LIN {X 0,Y 241.644,Z 1084.792,A -85,B 0,C 180,E1 20729.307,E2 20729.307} C_VEL
LIN {X 0,Y 219.298,Z 1111.875,A -85,B 0,C 180,E1 20736.62,E2 20736.62} C_VEL
LIN {X 0,Y 200.143,Z 1133.56,A -85,B 0,C 180,E1 20746.024,E2 20746.024} C_VEL
LIN {X 0,Y 185.27,Z 1150.433,A -85,B 0,C 180,E1 20757.915,E2 20757.915} C_VEL
LIN {X 0,Y 177.934,Z 1160.639,A -85,B 0,C 180,E1 20770.102,E2 20770.102} C_VEL
LIN {X 0,Y 175.677,Z 1165.283,A -85,B 0,C 180,E1 20780.076,E2 20780.076} C_VEL
LIN {X 0,Y 175.749,Z 1166.865,A -85,B 0,C 180,E1 20790.002,E2 20790.002} C_VEL
LIN {X 0,Y 175.679,Z 1165.296,A -85,B 0,C 180,E1 20799.928,E2 20799.928} C_VEL
LIN {X 0,Y 179.088,Z 1158.782,A -85,B 0,C 180,E1 20812.714,E2 20812.714} C_VEL
LIN {X 0,Y 187.491,Z 1147.762,A -85,B 0,C 180,E1 20824.426,E2 20824.426} C_VEL
LIN {X 0,Y 202.393,Z 1131.049,A -85,B 0,C 180,E1 20835.333,E2 20835.333} C_VEL
LIN {X 0,Y 222.783,Z 1108.004,A -85,B 0,C 180,E1 20844.647,E2 20844.647} C_VEL
LIN {X 0,Y 229.425,Z 1100.179,A -85,B 0,C 180,E1 20846.96,E2 20846.96} C_VEL
LIN {X 0,Y 230.286,Z 1098.317,A -85,B 0,C 180,E1 20847.685,E2 20847.685} C_VEL
LIN {X 0,Y 210.353,Z 1100.814,A -85,B 0,C 180,E1 20854.414,E2 20854.414} C_VEL
LIN {X 0,Y 197.119,Z 1101.191,A -85,B 0,C 180,E1 20862.106,E2 20862.106} C_VEL
LIN {X 0,Y 189.812,Z 1096.992,A -85,B 0,C 180,E1 20884.573,E2 20884.573} C_VEL
LIN {X 0,Y 207.688,Z 1091.37,A -85,B 0,C 180,E1 20901.373,E2 20901.373} C_VEL
LIN {X 0,Y 233.869,Z 1084.178,A -85,B 0,C 180,E1 20911.188,E2 20911.188} C_VEL
LIN {X 0,Y 240.479,Z 1082.186,A -85,B 0,C 180,E1 20912.869,E2 20912.869} C_VEL
LIN {X 0,Y 238.937,Z 1085.101,A -85,B 0,C 180,E1 20913.875,E2 20913.875} C_VEL
LIN {X 0,Y 235.19,Z 1089.54,A -85,B 0,C 180,E1 20914.966,E2 20914.966} C_VEL
LIN {X 0,Y 223.73,Z 1099.969,A -85,B 0,C 180,E1 20917.059,E2 20917.059} C_VEL
LIN {X 0,Y 212.332,Z 1109.522,A -85,B 0,C 180,E1 20919.465,E2 20919.465} C_VEL
LIN {X 0,Y 191.319,Z 1129.897,A -85,B 0,C 180,E1 20929.672,E2 20929.672} C_VEL
LIN {X 0,Y 176.864,Z 1143.663,A -85,B 0,C 180,E1 20941.908,E2 20941.908} C_VEL
LIN {X 0,Y 169.807,Z 1151.224,A -85,B 0,C 180,E1 20954.482,E2 20954.482} C_VEL
LIN {X 0,Y 167.781,Z 1154.034,A -85,B 0,C 180,E1 20964.82,E2 20964.82} C_VEL
LIN {X 0,Y 167.899,Z 1154.368,A -85,B 0,C 180,E1 20969.998,E2 20969.998} C_VEL
LIN {X 0,Y 168.419,Z 1152.942,A -85,B 0,C 180,E1 20980.356,E2 20980.356} C_VEL
LIN {X 0,Y 173.955,Z 1146.544,A -85,B 0,C 180,E1 20994.1,E2 20994.1} C_VEL
LIN {X 0,Y 185.565,Z 1135.234,A -85,B 0,C 180,E1 21006.266,E2 21006.266} C_VEL
LIN {X 0,Y 204.238,Z 1117.516,A -85,B 0,C 180,E1 21017.059,E2 21017.059} C_VEL
LIN {X 0,Y 226.928,Z 1093.954,A -85,B 0,C 180,E1 21025.462,E2 21025.462} C_VEL
LIN {X 0,Y 249.884,Z 1066.331,A -85,B 0,C 180,E1 21031.468,E2 21031.468} C_VEL
LIN {X 0,Y 271.022,Z 1035.748,A -85,B 0,C 180,E1 21035.688,E2 21035.688} C_VEL
LIN {X 0,Y 281.025,Z 1018.475,A -85,B 0,C 180,E1 21037.454,E2 21037.454} C_VEL
LIN {X 0,Y 280.826,Z 1004.794,A -85,B 0,C 180,E1 21043.501,E2 21043.501} C_VEL
LIN {X 0,Y 280.116,Z 996.302,A -85,B 0,C 180,E1 21049.097,E2 21049.097} C_VEL
LIN {X 0,Y 279.786,Z 992.242,A -85,B 0,C 180,E1 21053.789,E2 21053.789} C_VEL
LIN {X 0,Y 279.873,Z 990.81,A -85,B 0,C 180,E1 21056.901,E2 21056.901} C_VEL
LIN {X 0,Y 279.882,Z 991.061,A -85,B 0,C 180,E1 21060.001,E2 21060.001} C_VEL
LIN {X 0,Y 279.944,Z 995.928,A -85,B 0,C 180,E1 21066.211,E2 21066.211} C_VEL
LIN {X 0,Y 280.603,Z 1005.561,A -85,B 0,C 180,E1 21072.465,E2 21072.465} C_VEL
LIN {X 0,Y 280.581,Z 1019.974,A -85,B 0,C 180,E1 21078.553,E2 21078.553} C_VEL
LIN {X 0,Y 260.028,Z 1054.145,A -85,B 0,C 180,E1 21082.426,E2 21082.426} C_VEL
LIN {X 0,Y 237.05,Z 1085.261,A -85,B 0,C 180,E1 21087.757,E2 21087.757} C_VEL
LIN {X 0,Y 213.909,Z 1112.152,A -85,B 0,C 180,E1 21095.059,E2 21095.059} C_VEL
LIN {X 0,Y 193.525,Z 1133.989,A -85,B 0,C 180,E1 21104.757,E2 21104.757} C_VEL
LIN {X 0,Y 178.365,Z 1150.132,A -85,B 0,C 180,E1 21116.513,E2 21116.513} C_VEL
LIN {X 0,Y 170.325,Z 1160.341,A -85,B 0,C 180,E1 21129.173,E2 21129.173} C_VEL
LIN {X 0,Y 167.809,Z 1164.992,A -85,B 0,C 180,E1 21139.606,E2 21139.606} C_VEL
LIN {X 0,Y 167.84,Z 1166.578,A -85,B 0,C 180,E1 21150.002,E2 21150.002} C_VEL
LIN {X 0,Y 167.811,Z 1165.005,A -85,B 0,C 180,E1 21160.399,E2 21160.399} C_VEL
LIN {X 0,Y 171.429,Z 1158.708,A -85,B 0,C 180,E1 21173.422,E2 21173.422} C_VEL
LIN {X 0,Y 180.75,Z 1147.459,A -85,B 0,C 180,E1 21185.904,E2 21185.904} C_VEL
LIN {X 0,Y 197.204,Z 1130.076,A -85,B 0,C 180,E1 21197.406,E2 21197.406} C_VEL
LIN {X 0,Y 218.094,Z 1107.676,A -85,B 0,C 180,E1 21206.423,E2 21206.423} C_VEL
LIN {X 0,Y 220.393,Z 1105.118,A -85,B 0,C 180,E1 21207.202,E2 21207.202} C_VEL
LIN {X 0,Y 220.637,Z 1103.734,A -85,B 0,C 180,E1 21207.988,E2 21207.988} C_VEL
LIN {X 0,Y 197.119,Z 1105.708,A -85,B 0,C 180,E1 21217.415,E2 21217.415} C_VEL
LIN {X 0,Y 183.691,Z 1104.522,A -85,B 0,C 180,E1 21230.51,E2 21230.51} C_VEL
LIN {X 0,Y 195.152,Z 1097.977,A -85,B 0,C 180,E1 21258.076,E2 21258.076} C_VEL
LIN {X 0,Y 224.215,Z 1090.499,A -85,B 0,C 180,E1 21270.839,E2 21270.839} C_VEL
LIN {X 0,Y 230.972,Z 1088.637,A -85,B 0,C 180,E1 21272.665,E2 21272.665} C_VEL
LIN {X 0,Y 228.841,Z 1091.915,A -85,B 0,C 180,E1 21273.868,E2 21273.868} C_VEL
LIN {X 0,Y 212.332,Z 1109.522,A -85,B 0,C 180,E1 21279.465,E2 21279.465} C_VEL
LIN {X 0,Y 200.951,Z 1118.322,A -85,B 0,C 180,E1 21282.252,E2 21282.252} C_VEL
LIN {X 0,Y 189.711,Z 1126.107,A -85,B 0,C 180,E1 21285.477,E2 21285.477} C_VEL
LIN {X 0,Y 173.878,Z 1140.269,A -85,B 0,C 180,E1 21296.471,E2 21296.471} C_VEL
LIN {X 0,Y 163.142,Z 1150.371,A -85,B 0,C 180,E1 21311.042,E2 21311.042} C_VEL
LIN {X 0,Y 159.89,Z 1154.322,A -85,B 0,C 180,E1 21324.564,E2 21324.564} C_VEL
LIN {X 0,Y 160.014,Z 1154.655,A -85,B 0,C 180,E1 21329.997,E2 21329.997} C_VEL
LIN {X 0,Y 160.595,Z 1153.232,A -85,B 0,C 180,E1 21340.867,E2 21340.867} C_VEL
LIN {X 0,Y 165.989,Z 1147.48,A -85,B 0,C 180,E1 21354.212,E2 21354.212} C_VEL
LIN {X 0,Y 179.105,Z 1135.531,A -85,B 0,C 180,E1 21367.797,E2 21367.797} C_VEL
LIN {X 0,Y 198.827,Z 1117.825,A -85,B 0,C 180,E1 21378.762,E2 21378.762} C_VEL
LIN {X 0,Y 222.437,Z 1094.311,A -85,B 0,C 180,E1 21387.162,E2 21387.162} C_VEL
LIN {X 0,Y 246.18,Z 1066.68,A -85,B 0,C 180,E1 21393.1,E2 21393.1} C_VEL
LIN {X 0,Y 268.411,Z 1035.251,A -85,B 0,C 180,E1 21397.333,E2 21397.333} C_VEL
LIN {X 0,Y 276.139,Z 1022.065,A -85,B 0,C 180,E1 21398.768,E2 21398.768} C_VEL
LIN {X 0,Y 276.353,Z 1010.675,A -85,B 0,C 180,E1 21404.104,E2 21404.104} C_VEL
LIN {X 0,Y 276.075,Z 1001.74,A -85,B 0,C 180,E1 21410.532,E2 21410.532} C_VEL
LIN {X 0,Y 276.038,Z 997.771,A -85,B 0,C 180,E1 21416.857,E2 21416.857} C_VEL
LIN {X 0,Y 276.044,Z 998.005,A -85,B 0,C 180,E1 21420.001,E2 21420.001} C_VEL
LIN {X 0,Y 275.992,Z 1001.273,A -85,B 0,C 180,E1 21424.721,E2 21424.721} C_VEL
LIN {X 0,Y 276.129,Z 1009.965,A -85,B 0,C 180,E1 21431.065,E2 21431.065} C_VEL
LIN {X 0,Y 275.75,Z 1022.623,A -85,B 0,C 180,E1 21436.894,E2 21436.894} C_VEL
LIN {X 0,Y 274.36,Z 1026.277,A -85,B 0,C 180,E1 21437.626,E2 21437.626} C_VEL
LIN {X 0,Y 253.21,Z 1059.148,A -85,B 0,C 180,E1 21441.494,E2 21441.494} C_VEL
LIN {X 0,Y 229.95,Z 1088.949,A -85,B 0,C 180,E1 21446.873,E2 21446.873} C_VEL
LIN {X 0,Y 206.813,Z 1114.353,A -85,B 0,C 180,E1 21454.106,E2 21454.106} C_VEL
LIN {X 0,Y 187.223,Z 1134.23,A -85,B 0,C 180,E1 21463.296,E2 21463.296} C_VEL
LIN {X 0,Y 171.575,Z 1149.832,A -85,B 0,C 180,E1 21475,E2 21475} C_VEL
LIN {X 0,Y 162.558,Z 1160.344,A -85,B 0,C 180,E1 21488.649,E2 21488.649} C_VEL
LIN {X 0,Y 159.936,Z 1164.7,A -85,B 0,C 180,E1 21499.088,E2 21499.088} C_VEL
LIN {X 0,Y 159.952,Z 1166.291,A -85,B 0,C 180,E1 21510.003,E2 21510.003} C_VEL
LIN {X 0,Y 159.938,Z 1164.714,A -85,B 0,C 180,E1 21520.917,E2 21520.917} C_VEL
LIN {X 0,Y 163.981,Z 1158.411,A -85,B 0,C 180,E1 21534.554,E2 21534.554} C_VEL
LIN {X 0,Y 175.277,Z 1146.018,A -85,B 0,C 180,E1 21548.488,E2 21548.488} C_VEL
LIN {X 0,Y 193.018,Z 1128.453,A -85,B 0,C 180,E1 21559.896,E2 21559.896} C_VEL
LIN {X 0,Y 211.907,Z 1108.74,A -85,B 0,C 180,E1 21568.011,E2 21568.011} C_VEL
LIN {X 0,Y 191.121,Z 1110.194,A -85,B 0,C 180,E1 21576.665,E2 21576.665} C_VEL
LIN {X 0,Y 177.287,Z 1108.985,A -85,B 0,C 180,E1 21590.164,E2 21590.164} C_VEL
LIN {X 0,Y 188.974,Z 1102.525,A -85,B 0,C 180,E1 21618.688,E2 21618.688} C_VEL
LIN {X 0,Y 220.33,Z 1095.014,A -85,B 0,C 180,E1 21632.174,E2 21632.174} C_VEL
LIN {X 0,Y 221.641,Z 1094.669,A -85,B 0,C 180,E1 21632.539,E2 21632.539} C_VEL
LIN {X 0,Y 216.26,Z 1100.866,A -85,B 0,C 180,E1 21634.644,E2 21634.644} C_VEL
LIN {X 0,Y 195.481,Z 1120.888,A -85,B 0,C 180,E1 21642.619,E2 21642.619} C_VEL
LIN {X 0,Y 189.711,Z 1126.107,A -85,B 0,C 180,E1 21645.477,E2 21645.477} C_VEL
LIN {X 0,Y 178.917,Z 1133.074,A -85,B 0,C 180,E1 21649.213,E2 21649.213} C_VEL
LIN {X 0,Y 168.871,Z 1139.124,A -85,B 0,C 180,E1 21653.496,E2 21653.496} C_VEL
LIN {X 0,Y 156.972,Z 1149.324,A -85,B 0,C 180,E1 21667.302,E2 21667.302} C_VEL
LIN {X 0,Y 152.791,Z 1153.563,A -85,B 0,C 180,E1 21678.566,E2 21678.566} C_VEL
LIN {X 0,Y 152.109,Z 1154.943,A -85,B 0,C 180,E1 21689.997,E2 21689.997} C_VEL
LIN {X 0,Y 152.807,Z 1153.521,A -85,B 0,C 180,E1 21701.428,E2 21701.428} C_VEL
LIN {X 0,Y 158.677,Z 1147.773,A -85,B 0,C 180,E1 21715.405,E2 21715.405} C_VEL
LIN {X 0,Y 172.8,Z 1135.826,A -85,B 0,C 180,E1 21729.437,E2 21729.437} C_VEL
LIN {X 0,Y 193.586,Z 1118.135,A -85,B 0,C 180,E1 21740.564,E2 21740.564} C_VEL
LIN {X 0,Y 216.978,Z 1095.925,A -85,B 0,C 180,E1 21748.591,E2 21748.591} C_VEL
LIN {X 0,Y 241.184,Z 1068.925,A -85,B 0,C 180,E1 21754.478,E2 21754.478} C_VEL
LIN {X 0,Y 265.11,Z 1036.218,A -85,B 0,C 180,E1 21758.855,E2 21758.855} C_VEL
LIN {X 0,Y 271.302,Z 1026.26,A -85,B 0,C 180,E1 21759.911,E2 21759.911} C_VEL
LIN {X 0,Y 271.9,Z 1015.266,A -85,B 0,C 180,E1 21765.491,E2 21765.491} C_VEL
LIN {X 0,Y 271.963,Z 1007.356,A -85,B 0,C 180,E1 21771.841,E2 21771.841} C_VEL
LIN {X 0,Y 272.14,Z 1004.694,A -85,B 0,C 180,E1 21776.812,E2 21776.812} C_VEL
LIN {X 0,Y 272.132,Z 1004.931,A -85,B 0,C 180,E1 21780.002,E2 21780.002} C_VEL
LIN {X 0,Y 271.859,Z 1008.282,A -85,B 0,C 180,E1 21784.793,E2 21784.793} C_VEL
LIN {X 0,Y 271.688,Z 1017.25,A -85,B 0,C 180,E1 21791.248,E2 21791.248} C_VEL
LIN {X 0,Y 270.934,Z 1026.848,A -85,B 0,C 180,E1 21795.774,E2 21795.774} C_VEL
LIN {X 0,Y 269.441,Z 1030.146,A -85,B 0,C 180,E1 21796.386,E2 21796.386} C_VEL
LIN {X 0,Y 245.905,Z 1064.72,A -85,B 0,C 180,E1 21800.612,E2 21800.612} C_VEL
LIN {X 0,Y 221.132,Z 1094.468,A -85,B 0,C 180,E1 21806.369,E2 21806.369} C_VEL
LIN {X 0,Y 197.783,Z 1118.602,A -85,B 0,C 180,E1 21813.907,E2 21813.907} C_VEL
LIN {X 0,Y 175.552,Z 1139.532,A -85,B 0,C 180,E1 21824.984,E2 21824.984} C_VEL
LIN {X 0,Y 160.652,Z 1153.722,A -85,B 0,C 180,E1 21838.014,E2 21838.014} C_VEL
LIN {X 0,Y 153.249,Z 1162.465,A -85,B 0,C 180,E1 21852.761,E2 21852.761} C_VEL
LIN {X 0,Y 151.723,Z 1165.758,A -85,B 0,C 180,E1 21866.268,E2 21866.268} C_VEL
LIN {X 0,Y 151.718,Z 1165.763,A -85,B 0,C 180,E1 21873.704,E2 21873.704} C_VEL
LIN {X 0,Y 153.245,Z 1162.485,A -85,B 0,C 180,E1 21887.245,E2 21887.245} C_VEL
LIN {X 0,Y 160.574,Z 1153.797,A -85,B 0,C 180,E1 21901.941,E2 21901.941} C_VEL
LIN {X 0,Y 176.95,Z 1138.345,A -85,B 0,C 180,E1 21915.91,E2 21915.91} C_VEL
LIN {X 0,Y 199.316,Z 1117.193,A -85,B 0,C 180,E1 21926.685,E2 21926.685} C_VEL
LIN {X 0,Y 201.855,Z 1114.63,A -85,B 0,C 180,E1 21927.628,E2 21927.628} C_VEL
LIN {X 0,Y 202.05,Z 1113.567,A -85,B 0,C 180,E1 21928.363,E2 21928.363} C_VEL
LIN {X 0,Y 178.552,Z 1114.416,A -85,B 0,C 180,E1 21940.172,E2 21940.172} C_VEL
LIN {X 0,Y 170.346,Z 1110.449,A -85,B 0,C 180,E1 21965.096,E2 21965.096} C_VEL
LIN {X 0,Y 189.781,Z 1105.392,A -85,B 0,C 180,E1 21983.505,E2 21983.505} C_VEL
LIN {X 0,Y 212.145,Z 1100.335,A -85,B 0,C 180,E1 21992.357,E2 21992.357} C_VEL
LIN {X 0,Y 205.427,Z 1107.331,A -85,B 0,C 180,E1 21994.913,E2 21994.913} C_VEL
LIN {X 0,Y 183.207,Z 1127.096,A -85,B 0,C 180,E1 22004.142,E2 22004.142} C_VEL
LIN {X 0,Y 168.871,Z 1139.124,A -85,B 0,C 180,E1 22013.496,E2 22013.496} C_VEL
LIN {X 0,Y 159.567,Z 1144.315,A -85,B 0,C 180,E1 22018.35,E2 22018.35} C_VEL
LIN {X 0,Y 151.045,Z 1148.424,A -85,B 0,C 180,E1 22023.826,E2 22023.826} C_VEL
LIN {X 0,Y 144.991,Z 1153.852,A -85,B 0,C 180,E1 22037.942,E2 22037.942} C_VEL
LIN {X 0,Y 144.223,Z 1155.229,A -85,B 0,C 180,E1 22049.997,E2 22049.997} C_VEL
LIN {X 0,Y 145.007,Z 1153.811,A -85,B 0,C 180,E1 22062.051,E2 22062.051} C_VEL
LIN {X 0,Y 151.653,Z 1147.918,A -85,B 0,C 180,E1 22076.989,E2 22076.989} C_VEL
LIN {X 0,Y 166.627,Z 1136.122,A -85,B 0,C 180,E1 22091.206,E2 22091.206} C_VEL
LIN {X 0,Y 188.564,Z 1118.444,A -85,B 0,C 180,E1 22102.458,E2 22102.458} C_VEL
LIN {X 0,Y 213.132,Z 1096.032,A -85,B 0,C 180,E1 22110.486,E2 22110.486} C_VEL
LIN {X 0,Y 237.844,Z 1069.278,A -85,B 0,C 180,E1 22116.219,E2 22116.219} C_VEL
LIN {X 0,Y 262.354,Z 1036.632,A -85,B 0,C 180,E1 22120.471,E2 22120.471} C_VEL
LIN {X 0,Y 266.078,Z 1030.821,A -85,B 0,C 180,E1 22121.06,E2 22121.06} C_VEL
LIN {X 0,Y 267.196,Z 1022.422,A -85,B 0,C 180,E1 22125.228,E2 22125.228} C_VEL
LIN {X 0,Y 267.649,Z 1015.15,A -85,B 0,C 180,E1 22130.856,E2 22130.856} C_VEL
LIN {X 0,Y 267.965,Z 1011.478,A -85,B 0,C 180,E1 22136.763,E2 22136.763} C_VEL
LIN {X 0,Y 267.96,Z 1011.701,A -85,B 0,C 180,E1 22140.002,E2 22140.002} C_VEL
LIN {X 0,Y 267.605,Z 1015.21,A -85,B 0,C 180,E1 22144.87,E2 22144.87} C_VEL
LIN {X 0,Y 266.974,Z 1023.501,A -85,B 0,C 180,E1 22150.929,E2 22150.929} C_VEL
LIN {X 0,Y 266.102,Z 1031.174,A -85,B 0,C 180,E1 22154.697,E2 22154.697} C_VEL
LIN {X 0,Y 242.75,Z 1064.854,A -85,B 0,C 180,E1 22158.886,E2 22158.886} C_VEL
LIN {X 0,Y 218.067,Z 1093.663,A -85,B 0,C 180,E1 22164.315,E2 22164.315} C_VEL
LIN {X 0,Y 192.416,Z 1119.042,A -85,B 0,C 180,E1 22172.174,E2 22172.174} C_VEL
LIN {X 0,Y 169.699,Z 1139.331,A -85,B 0,C 180,E1 22183.093,E2 22183.093} C_VEL
LIN {X 0,Y 153.74,Z 1153.422,A -85,B 0,C 180,E1 22196.391,E2 22196.391} C_VEL
LIN {X 0,Y 145.561,Z 1162.17,A -85,B 0,C 180,E1 22211.819,E2 22211.819} C_VEL
LIN {X 0,Y 143.859,Z 1165.301,A -85,B 0,C 180,E1 22223.961,E2 22223.961} C_VEL
LIN {X 0,Y 144.131,Z 1165.715,A -85,B 0,C 180,E1 22230.003,E2 22230.003} C_VEL
LIN {X 0,Y 144.251,Z 1164.131,A -85,B 0,C 180,E1 22242.121,E2 22242.121} C_VEL
LIN {X 0,Y 149.268,Z 1157.818,A -85,B 0,C 180,E1 22257.162,E2 22257.162} C_VEL
LIN {X 0,Y 163.132,Z 1145.033,A -85,B 0,C 180,E1 22272.453,E2 22272.453} C_VEL
LIN {X 0,Y 183.964,Z 1126.83,A -85,B 0,C 180,E1 22284.371,E2 22284.371} C_VEL
LIN {X 0,Y 193.248,Z 1118.033,A -85,B 0,C 180,E1 22288.453,E2 22288.453} C_VEL
LIN {X 0,Y 172.215,Z 1118.514,A -85,B 0,C 180,E1 22299.41,E2 22299.41} C_VEL
LIN {X 0,Y 163.682,Z 1114.676,A -85,B 0,C 180,E1 22325.305,E2 22325.305} C_VEL
LIN {X 0,Y 183.63,Z 1109.654,A -85,B 0,C 180,E1 22344.342,E2 22344.342} C_VEL
LIN {X 0,Y 202.445,Z 1105.782,A -85,B 0,C 180,E1 22352.09,E2 22352.09} C_VEL
LIN {X 0,Y 197.776,Z 1110.528,A -85,B 0,C 180,E1 22354.089,E2 22354.089} C_VEL
LIN {X 0,Y 174.447,Z 1130.026,A -85,B 0,C 180,E1 22363.967,E2 22363.967} C_VEL
LIN {X 0,Y 155.967,Z 1144.538,A -85,B 0,C 180,E1 22377.725,E2 22377.725} C_VEL
LIN {X 0,Y 151.045,Z 1148.424,A -85,B 0,C 180,E1 22383.826,E2 22383.826} C_VEL
LIN {X 0,Y 145.742,Z 1150.941,A -85,B 0,C 180,E1 22388.377,E2 22388.377} C_VEL
LIN {X 0,Y 137.671,Z 1153.725,A -85,B 0,C 180,E1 22395.637,E2 22395.637} C_VEL
LIN {X 0,Y 137.375,Z 1153.945,A -85,B 0,C 180,E1 22396.54,E2 22396.54} C_VEL
LIN {X 0,Y 136.258,Z 1155.485,A -85,B 0,C 180,E1 22410.712,E2 22410.712} C_VEL
LIN {X 0,Y 137.249,Z 1154.1,A -85,B 0,C 180,E1 22422.744,E2 22422.744} C_VEL
LIN {X 0,Y 144.325,Z 1148.347,A -85,B 0,C 180,E1 22438.168,E2 22438.168} C_VEL
LIN {X 0,Y 160.651,Z 1136.417,A -85,B 0,C 180,E1 22453.099,E2 22453.099} C_VEL
LIN {X 0,Y 183.764,Z 1118.751,A -85,B 0,C 180,E1 22464.451,E2 22464.451} C_VEL
LIN {X 0,Y 209.282,Z 1096.357,A -85,B 0,C 180,E1 22472.405,E2 22472.405} C_VEL
LIN {X 0,Y 236.294,Z 1067.752,A -85,B 0,C 180,E1 22478.296,E2 22478.296} C_VEL
LIN {X 0,Y 259.974,Z 1036.785,A -85,B 0,C 180,E1 22482.15,E2 22482.15} C_VEL
LIN {X 0,Y 261.734,Z 1033.582,A -85,B 0,C 180,E1 22482.733,E2 22482.733} C_VEL
LIN {X 0,Y 262.888,Z 1024.664,A -85,B 0,C 180,E1 22488.267,E2 22488.267} C_VEL
LIN {X 0,Y 263.374,Z 1019.737,A -85,B 0,C 180,E1 22493.4,E2 22493.4} C_VEL
LIN {X 0,Y 263.681,Z 1018.2,A -85,B 0,C 180,E1 22496.71,E2 22496.71} C_VEL
LIN {X 0,Y 263.425,Z 1019.36,A -85,B 0,C 180,E1 22501.648,E2 22501.648} C_VEL
LIN {X 0,Y 262.76,Z 1024.969,A -85,B 0,C 180,E1 22507.5,E2 22507.5} C_VEL
LIN {X 0,Y 261.342,Z 1035.053,A -85,B 0,C 180,E1 22513.4,E2 22513.4} C_VEL
LIN {X 0,Y 238.035,Z 1067.14,A -85,B 0,C 180,E1 22517.424,E2 22517.424} C_VEL
LIN {X 0,Y 213.32,Z 1094.826,A -85,B 0,C 180,E1 22522.676,E2 22522.676} C_VEL
LIN {X 0,Y 186.755,Z 1119.907,A -85,B 0,C 180,E1 22530.527,E2 22530.527} C_VEL
LIN {X 0,Y 164.775,Z 1138.545,A -85,B 0,C 180,E1 22540.626,E2 22540.626} C_VEL
LIN {X 0,Y 147.028,Z 1153.075,A -85,B 0,C 180,E1 22554.55,E2 22554.55} C_VEL
LIN {X 0,Y 137.897,Z 1161.874,A -85,B 0,C 180,E1 22570.77,E2 22570.77} C_VEL
LIN {X 0,Y 135.941,Z 1165.011,A -85,B 0,C 180,E1 22583.608,E2 22583.608} C_VEL
LIN {X 0,Y 136.224,Z 1165.428,A -85,B 0,C 180,E1 22590.003,E2 22590.003} C_VEL
LIN {X 0,Y 136.441,Z 1163.84,A -85,B 0,C 180,E1 22602.826,E2 22602.826} C_VEL
LIN {X 0,Y 142.042,Z 1157.521,A -85,B 0,C 180,E1 22618.668,E2 22618.668} C_VEL
LIN {X 0,Y 156.97,Z 1144.854,A -85,B 0,C 180,E1 22634.377,E2 22634.377} C_VEL
LIN {X 0,Y 179.286,Z 1126.524,A -85,B 0,C 180,E1 22646.514,E2 22646.514} C_VEL
LIN {X 0,Y 183.295,Z 1123.091,A -85,B 0,C 180,E1 22648.123,E2 22648.123} C_VEL
LIN {X 0,Y 183.254,Z 1122.24,A -85,B 0,C 180,E1 22648.937,E2 22648.937} C_VEL
LIN {X 0,Y 165.841,Z 1122.45,A -85,B 0,C 180,E1 22658.58,E2 22658.58} C_VEL
LIN {X 0,Y 156.84,Z 1118.617,A -85,B 0,C 180,E1 22685.537,E2 22685.537} C_VEL
LIN {X 0,Y 177.462,Z 1113.837,A -85,B 0,C 180,E1 22705.247,E2 22705.247} C_VEL
LIN {X 0,Y 192.56,Z 1110.89,A -85,B 0,C 180,E1 22711.716,E2 22711.716} C_VEL
LIN {X 0,Y 192.376,Z 1111.72,A -85,B 0,C 180,E1 22712.433,E2 22712.433} C_VEL
LIN {X 0,Y 168.92,Z 1130.325,A -85,B 0,C 180,E1 22721.988,E2 22721.988} C_VEL
LIN {X 0,Y 149.207,Z 1144.829,A -85,B 0,C 180,E1 22736.07,E2 22736.07} C_VEL
LIN {X 0,Y 139.227,Z 1152.387,A -85,B 0,C 180,E1 22750.955,E2 22750.955} C_VEL
LIN {X 0,Y 137.375,Z 1153.945,A -85,B 0,C 180,E1 22756.54,E2 22756.54} C_VEL
LIN {X 0,Y 134.195,Z 1155.172,A -85,B 0,C 180,E1 22761.862,E2 22761.862} C_VEL
LIN {X 0,Y 128.298,Z 1155.741,A -85,B 0,C 180,E1 22771.193,E2 22771.193} C_VEL
LIN {X 0,Y 129.483,Z 1154.391,A -85,B 0,C 180,E1 22783.522,E2 22783.522} C_VEL
LIN {X 0,Y 137.298,Z 1148.638,A -85,B 0,C 180,E1 22799.75,E2 22799.75} C_VEL
LIN {X 0,Y 154.859,Z 1136.711,A -85,B 0,C 180,E1 22815.139,E2 22815.139} C_VEL
LIN {X 0,Y 179.175,Z 1119.071,A -85,B 0,C 180,E1 22826.545,E2 22826.545} C_VEL
LIN {X 0,Y 205.687,Z 1096.678,A -85,B 0,C 180,E1 22834.387,E2 22834.387} C_VEL
LIN {X 0,Y 233.46,Z 1068.108,A -85,B 0,C 180,E1 22840.116,E2 22840.116} C_VEL
LIN {X 0,Y 256.148,Z 1039.351,A -85,B 0,C 180,E1 22843.619,E2 22843.619} C_VEL
LIN {X 0,Y 257.272,Z 1036.157,A -85,B 0,C 180,E1 22844.937,E2 22844.937} C_VEL
LIN {X 0,Y 258.598,Z 1028.057,A -85,B 0,C 180,E1 22851.225,E2 22851.225} C_VEL
LIN {X 0,Y 259.203,Z 1024.791,A -85,B 0,C 180,E1 22856.653,E2 22856.653} C_VEL
LIN {X 0,Y 258.938,Z 1025.959,A -85,B 0,C 180,E1 22861.677,E2 22861.677} C_VEL
LIN {X 0,Y 257.949,Z 1031.767,A -85,B 0,C 180,E1 22867.641,E2 22867.641} C_VEL
LIN {X 0,Y 256.619,Z 1039.166,A -85,B 0,C 180,E1 22872.127,E2 22872.127} C_VEL
LIN {X 0,Y 230.807,Z 1072.625,A -85,B 0,C 180,E1 22876.383,E2 22876.383} C_VEL
LIN {X 0,Y 202.184,Z 1102.288,A -85,B 0,C 180,E1 22882.519,E2 22882.519} C_VEL
LIN {X 0,Y 176.107,Z 1125.128,A -85,B 0,C 180,E1 22890.713,E2 22890.713} C_VEL
LIN {X 0,Y 153.14,Z 1143.08,A -85,B 0,C 180,E1 22902.141,E2 22902.141} C_VEL
LIN {X 0,Y 137.133,Z 1155.342,A -85,B 0,C 180,E1 22916.495,E2 22916.495} C_VEL
LIN {X 0,Y 130.276,Z 1161.579,A -85,B 0,C 180,E1 22929.597,E2 22929.597} C_VEL
LIN {X 0,Y 128.025,Z 1164.721,A -85,B 0,C 180,E1 22943.211,E2 22943.211} C_VEL
LIN {X 0,Y 128.306,Z 1165.14,A -85,B 0,C 180,E1 22950.003,E2 22950.003} C_VEL
LIN {X 0,Y 128.618,Z 1163.548,A -85,B 0,C 180,E1 22963.621,E2 22963.621} C_VEL
LIN {X 0,Y 134.913,Z 1157.224,A -85,B 0,C 180,E1 22980.337,E2 22980.337} C_VEL
LIN {X 0,Y 151.173,Z 1144.553,A -85,B 0,C 180,E1 22996.569,E2 22996.569} C_VEL
LIN {X 0,Y 174.433,Z 1126.543,A -85,B 0,C 180,E1 23008.614,E2 23008.614} C_VEL
LIN {X 0,Y 154.271,Z 1125.622,A -85,B 0,C 180,E1 23022.875,E2 23022.875} C_VEL
LIN {X 0,Y 153.206,Z 1121.412,A -85,B 0,C 180,E1 23051.396,E2 23051.396} C_VEL
LIN {X 0,Y 171.225,Z 1117.791,A -85,B 0,C 180,E1 23066.235,E2 23066.235} C_VEL
LIN {X 0,Y 182.27,Z 1115.762,A -85,B 0,C 180,E1 23071.198,E2 23071.198} C_VEL
LIN {X 0,Y 182.625,Z 1116.389,A -85,B 0,C 180,E1 23072.146,E2 23072.146} C_VEL
LIN {X 0,Y 158.895,Z 1133.922,A -85,B 0,C 180,E1 23082.392,E2 23082.392} C_VEL
LIN {X 0,Y 142.581,Z 1145.121,A -85,B 0,C 180,E1 23094.259,E2 23094.259} C_VEL
LIN {X 0,Y 131.684,Z 1152.678,A -85,B 0,C 180,E1 23109.818,E2 23109.818} C_VEL
LIN {X 0,Y 128.377,Z 1155.474,A -85,B 0,C 180,E1 23123.223,E2 23123.223} C_VEL
LIN {X 0,Y 128.298,Z 1155.741,A -85,B 0,C 180,E1 23131.193,E2 23131.193} C_VEL
LIN {X 0,Y 125.785,Z 1155.535,A -85,B 0,C 180,E1 23136.986,E2 23136.986} C_VEL
LIN {X 0,Y 122.447,Z 1154.032,A -85,B 0,C 180,E1 23147.017,E2 23147.017} C_VEL
LIN {X 0,Y 133.117,Z 1147.171,A -85,B 0,C 180,E1 23164.658,E2 23164.658} C_VEL
LIN {X 0,Y 151.378,Z 1135.596,A -85,B 0,C 180,E1 23178.562,E2 23178.562} C_VEL
LIN {X 0,Y 176.224,Z 1118.308,A -85,B 0,C 180,E1 23189.223,E2 23189.223} C_VEL
LIN {X 0,Y 203.882,Z 1095.574,A -85,B 0,C 180,E1 23196.78,E2 23196.78} C_VEL
LIN {X 0,Y 230.869,Z 1068.465,A -85,B 0,C 180,E1 23201.978,E2 23201.978} C_VEL
LIN {X 0,Y 251.719,Z 1042.808,A -85,B 0,C 180,E1 23205.05,E2 23205.05} C_VEL
LIN {X 0,Y 253.47,Z 1036.026,A -85,B 0,C 180,E1 23209.679,E2 23209.679} C_VEL
LIN {X 0,Y 254.084,Z 1032.936,A -85,B 0,C 180,E1 23213.158,E2 23213.158} C_VEL
LIN {X 0,Y 254.563,Z 1031.265,A -85,B 0,C 180,E1 23216.592,E2 23216.592} C_VEL
LIN {X 0,Y 254.239,Z 1032.428,A -85,B 0,C 180,E1 23221.708,E2 23221.708} C_VEL
LIN {X 0,Y 252.966,Z 1038.437,A -85,B 0,C 180,E1 23227.74,E2 23227.74} C_VEL
LIN {X 0,Y 251.995,Z 1042.528,A -85,B 0,C 180,E1 23230.385,E2 23230.385} C_VEL
LIN {X 0,Y 249.541,Z 1046.419,A -85,B 0,C 180,E1 23231.189,E2 23231.189} C_VEL
LIN {X 0,Y 223.649,Z 1077.645,A -85,B 0,C 180,E1 23235.267,E2 23235.267} C_VEL
LIN {X 0,Y 196.871,Z 1104,A -85,B 0,C 180,E1 23240.89,E2 23240.89} C_VEL
LIN {X 0,Y 169.43,Z 1126.757,A -85,B 0,C 180,E1 23249.298,E2 23249.298} C_VEL
LIN {X 0,Y 145.622,Z 1144.194,A -85,B 0,C 180,E1 23261.081,E2 23261.081} C_VEL
LIN {X 0,Y 127.924,Z 1156.897,A -85,B 0,C 180,E1 23277.821,E2 23277.821} C_VEL
LIN {X 0,Y 120.817,Z 1163.238,A -85,B 0,C 180,E1 23295.487,E2 23295.487} C_VEL
LIN {X 0,Y 120.406,Z 1164.853,A -85,B 0,C 180,E1 23310.003,E2 23310.003} C_VEL
LIN {X 0,Y 120.816,Z 1163.255,A -85,B 0,C 180,E1 23324.519,E2 23324.519} C_VEL
LIN {X 0,Y 127.908,Z 1156.928,A -85,B 0,C 180,E1 23342.191,E2 23342.191} C_VEL
LIN {X 0,Y 145.629,Z 1144.254,A -85,B 0,C 180,E1 23358.924,E2 23358.924} C_VEL
LIN {X 0,Y 163.38,Z 1131.479,A -85,B 0,C 180,E1 23368.273,E2 23368.273} C_VEL
LIN {X 0,Y 164.707,Z 1130.053,A -85,B 0,C 180,E1 23369.319,E2 23369.319} C_VEL
LIN {X 0,Y 143.724,Z 1128.644,A -85,B 0,C 180,E1 23387.835,E2 23387.835} C_VEL
LIN {X 0,Y 157.204,Z 1122.921,A -85,B 0,C 180,E1 23422.654,E2 23422.654} C_VEL
LIN {X 0,Y 173.809,Z 1120.209,A -85,B 0,C 180,E1 23431.506,E2 23431.506} C_VEL
LIN {X 0,Y 149.057,Z 1137.19,A -85,B 0,C 180,E1 23442.673,E2 23442.673} C_VEL
LIN {X 0,Y 130.342,Z 1148.999,A -85,B 0,C 180,E1 23458.48,E2 23458.48} C_VEL
LIN {X 0,Y 121.746,Z 1154.72,A -85,B 0,C 180,E1 23475.594,E2 23475.594} C_VEL
LIN {X 0,Y 120.411,Z 1156.04,A -85,B 0,C 180,E1 23491.036,E2 23491.036} C_VEL
LIN {X 0,Y 122.447,Z 1154.032,A -85,B 0,C 180,E1 23507.017,E2 23507.017} C_VEL
LIN {X 0,Y 122.691,Z 1153.159,A -85,B 0,C 180,E1 23511.08,E2 23511.08} C_VEL
LIN {X 0,Y 122.738,Z 1149.711,A -85,B 0,C 180,E1 23522.338,E2 23522.338} C_VEL
LIN {X 0,Y 123.43,Z 1149.297,A -85,B 0,C 180,E1 23523.294,E2 23523.294} C_VEL
LIN {X 0,Y 143.488,Z 1137.543,A -85,B 0,C 180,E1 23539.47,E2 23539.47} C_VEL
LIN {X 0,Y 169.435,Z 1120.611,A -85,B 0,C 180,E1 23550.623,E2 23550.623} C_VEL
LIN {X 0,Y 199.278,Z 1097.316,A -85,B 0,C 180,E1 23558.549,E2 23558.549} C_VEL
LIN {X 0,Y 228.517,Z 1068.823,A -85,B 0,C 180,E1 23563.889,E2 23563.889} C_VEL
LIN {X 0,Y 246.642,Z 1047.361,A -85,B 0,C 180,E1 23566.409,E2 23566.409} C_VEL
LIN {X 0,Y 247.798,Z 1044.586,A -85,B 0,C 180,E1 23567.858,E2 23567.858} C_VEL
LIN {X 0,Y 249.222,Z 1039.424,A -85,B 0,C 180,E1 23573.023,E2 23573.023} C_VEL
LIN {X 0,Y 249.787,Z 1037.656,A -85,B 0,C 180,E1 23576.527,E2 23576.527} C_VEL
LIN {X 0,Y 249.443,Z 1038.838,A -85,B 0,C 180,E1 23581.741,E2 23581.741} C_VEL
LIN {X 0,Y 247.687,Z 1045.149,A -85,B 0,C 180,E1 23588.002,E2 23588.002} C_VEL
LIN {X 0,Y 246.608,Z 1047.993,A -85,B 0,C 180,E1 23589.538,E2 23589.538} C_VEL
LIN {X 0,Y 219.943,Z 1079.079,A -85,B 0,C 180,E1 23593.501,E2 23593.501} C_VEL
LIN {X 0,Y 190.637,Z 1106.643,A -85,B 0,C 180,E1 23599.415,E2 23599.415} C_VEL
LIN {X 0,Y 161.671,Z 1129.243,A -85,B 0,C 180,E1 23608.198,E2 23608.198} C_VEL
LIN {X 0,Y 136.009,Z 1146.727,A -85,B 0,C 180,E1 23621.374,E2 23621.374} C_VEL
LIN {X 0,Y 118.74,Z 1158.255,A -85,B 0,C 180,E1 23639.336,E2 23639.336} C_VEL
LIN {X 0,Y 113.046,Z 1162.945,A -85,B 0,C 180,E1 23654.466,E2 23654.466} C_VEL
LIN {X 0,Y 112.484,Z 1164.565,A -85,B 0,C 180,E1 23670.004,E2 23670.004} C_VEL
LIN {X 0,Y 113.045,Z 1162.963,A -85,B 0,C 180,E1 23685.542,E2 23685.542} C_VEL
LIN {X 0,Y 120.982,Z 1156.689,A -85,B 0,C 180,E1 23704.132,E2 23704.132} C_VEL
LIN {X 0,Y 140.326,Z 1143.952,A -85,B 0,C 180,E1 23721.475,E2 23721.475} C_VEL
LIN {X 0,Y 155.445,Z 1133.359,A -85,B 0,C 180,E1 23729.761,E2 23729.761} C_VEL
LIN {X 0,Y 136.775,Z 1132.014,A -85,B 0,C 180,E1 23747.207,E2 23747.207} C_VEL
LIN {X 0,Y 150.735,Z 1126.53,A -85,B 0,C 180,E1 23783.685,E2 23783.685} C_VEL
LIN {X 0,Y 163.206,Z 1124.517,A -85,B 0,C 180,E1 23790.714,E2 23790.714} C_VEL
LIN {X 0,Y 158.451,Z 1128.127,A -85,B 0,C 180,E1 23793.261,E2 23793.261} C_VEL
LIN {X 0,Y 135.347,Z 1142.434,A -85,B 0,C 180,E1 23805.634,E2 23805.634} C_VEL
LIN {X 0,Y 118.975,Z 1151.948,A -85,B 0,C 180,E1 23822.959,E2 23822.959} C_VEL
LIN {X 0,Y 112.649,Z 1156.05,A -85,B 0,C 180,E1 23842.272,E2 23842.272} C_VEL
LIN {X 0,Y 112.621,Z 1156.379,A -85,B 0,C 180,E1 23849.996,E2 23849.996} C_VEL
LIN {X 0,Y 114.645,Z 1154.458,A -85,B 0,C 180,E1 23867.607,E2 23867.607} C_VEL
LIN {X 0,Y 123.43,Z 1149.297,A -85,B 0,C 180,E1 23883.294,E2 23883.294} C_VEL
LIN {X 0,Y 125.592,Z 1147.598,A -85,B 0,C 180,E1 23887.118,E2 23887.118} C_VEL
LIN {X 0,Y 130.787,Z 1142.125,A -85,B 0,C 180,E1 23897.444,E2 23897.444} C_VEL
LIN {X 0,Y 131.88,Z 1141.491,A -85,B 0,C 180,E1 23898.233,E2 23898.233} C_VEL
LIN {X 0,Y 158.734,Z 1125.496,A -85,B 0,C 180,E1 23910.767,E2 23910.767} C_VEL
LIN {X 0,Y 187.521,Z 1104.917,A -85,B 0,C 180,E1 23918.848,E2 23918.848} C_VEL
LIN {X 0,Y 216.781,Z 1079.09,A -85,B 0,C 180,E1 23924.379,E2 23924.379} C_VEL
LIN {X 0,Y 242.055,Z 1051.287,A -85,B 0,C 180,E1 23927.883,E2 23927.883} C_VEL
LIN {X 0,Y 243.563,Z 1047.279,A -85,B 0,C 180,E1 23931.081,E2 23931.081} C_VEL
LIN {X 0,Y 244.775,Z 1043.899,A -85,B 0,C 180,E1 23936.456,E2 23936.456} C_VEL
LIN {X 0,Y 244.81,Z 1044.029,A -85,B 0,C 180,E1 23940.002,E2 23940.002} C_VEL
LIN {X 0,Y 243.053,Z 1049.254,A -85,B 0,C 180,E1 23946.291,E2 23946.291} C_VEL
LIN {X 0,Y 242.504,Z 1051.062,A -85,B 0,C 180,E1 23947.686,E2 23947.686} C_VEL
LIN {X 0,Y 239.503,Z 1054.951,A -85,B 0,C 180,E1 23948.387,E2 23948.387} C_VEL
LIN {X 0,Y 212.198,Z 1084.683,A -85,B 0,C 180,E1 23952.361,E2 23952.361} C_VEL
LIN {X 0,Y 183.279,Z 1110.239,A -85,B 0,C 180,E1 23958.192,E2 23958.192} C_VEL
LIN {X 0,Y 153.3,Z 1132.066,A -85,B 0,C 180,E1 23967.267,E2 23967.267} C_VEL
LIN {X 0,Y 128.949,Z 1147.522,A -85,B 0,C 180,E1 23979.827,E2 23979.827} C_VEL
LIN {X 0,Y 111.784,Z 1157.956,A -85,B 0,C 180,E1 23997.197,E2 23997.197} C_VEL
LIN {X 0,Y 105.321,Z 1162.652,A -85,B 0,C 180,E1 24013.294,E2 24013.294} C_VEL
LIN {X 0,Y 104.56,Z 1164.276,A -85,B 0,C 180,E1 24030.004,E2 24030.004} C_VEL
LIN {X 0,Y 105.321,Z 1162.671,A -85,B 0,C 180,E1 24046.714,E2 24046.714} C_VEL
LIN {X 0,Y 113.67,Z 1156.773,A -85,B 0,C 180,E1 24065.585,E2 24065.585} C_VEL
LIN {X 0,Y 133.012,Z 1145.044,A -85,B 0,C 180,E1 24082.835,E2 24082.835} C_VEL
LIN {X 0,Y 144.594,Z 1137.861,A -85,B 0,C 180,E1 24089.016,E2 24089.016} C_VEL
LIN {X 0,Y 145.652,Z 1136.581,A -85,B 0,C 180,E1 24090.514,E2 24090.514} C_VEL
LIN {X 0,Y 127.591,Z 1134.537,A -85,B 0,C 180,E1 24113.182,E2 24113.182} C_VEL
LIN {X 0,Y 152.465,Z 1128.604,A -85,B 0,C 180,E1 24149.765,E2 24149.765} C_VEL
LIN {X 0,Y 153.62,Z 1128.439,A -85,B 0,C 180,E1 24150.359,E2 24150.359} C_VEL
LIN {X 0,Y 148.104,Z 1132.216,A -85,B 0,C 180,E1 24153.191,E2 24153.191} C_VEL
LIN {X 0,Y 125.035,Z 1145.269,A -85,B 0,C 180,E1 24166.588,E2 24166.588} C_VEL
LIN {X 0,Y 109.451,Z 1153.55,A -85,B 0,C 180,E1 24185.476,E2 24185.476} C_VEL
LIN {X 0,Y 104.803,Z 1156.338,A -85,B 0,C 180,E1 24201.689,E2 24201.689} C_VEL
LIN {X 0,Y 104.727,Z 1156.666,A -85,B 0,C 180,E1 24209.996,E2 24209.996} C_VEL
LIN {X 0,Y 106.373,Z 1155.262,A -85,B 0,C 180,E1 24226.536,E2 24226.536} C_VEL
LIN {X 0,Y 116.952,Z 1149.515,A -85,B 0,C 180,E1 24245.629,E2 24245.629} C_VEL
LIN {X 0,Y 131.88,Z 1141.491,A -85,B 0,C 180,E1 24258.233,E2 24258.233} C_VEL
LIN {X 0,Y 138.671,Z 1136.577,A -85,B 0,C 180,E1 24264.773,E2 24264.773} C_VEL
LIN {X 0,Y 146.832,Z 1130.649,A -85,B 0,C 180,E1 24270.532,E2 24270.532} C_VEL
LIN {X 0,Y 176.058,Z 1111.649,A -85,B 0,C 180,E1 24279.265,E2 24279.265} C_VEL
LIN {X 0,Y 205.738,Z 1087.8,A -85,B 0,C 180,E1 24285.05,E2 24285.05} C_VEL
LIN {X 0,Y 234.589,Z 1058.603,A -85,B 0,C 180,E1 24289.06,E2 24289.06} C_VEL
LIN {X 0,Y 237.666,Z 1054.939,A -85,B 0,C 180,E1 24289.494,E2 24289.494} C_VEL
LIN {X 0,Y 238.797,Z 1052.006,A -85,B 0,C 180,E1 24292.717,E2 24292.717} C_VEL
LIN {X 0,Y 239.69,Z 1050.091,A -85,B 0,C 180,E1 24296.38,E2 24296.38} C_VEL
LIN {X 0,Y 239.742,Z 1050.192,A -85,B 0,C 180,E1 24300.002,E2 24300.002} C_VEL
LIN {X 0,Y 237.538,Z 1055.568,A -85,B 0,C 180,E1 24306.441,E2 24306.441} C_VEL
LIN {X 0,Y 209.473,Z 1085.393,A -85,B 0,C 180,E1 24310.354,E2 24310.354} C_VEL
LIN {X 0,Y 179.225,Z 1111.155,A -85,B 0,C 180,E1 24316.065,E2 24316.065} C_VEL
LIN {X 0,Y 149.698,Z 1131.76,A -85,B 0,C 180,E1 24324.458,E2 24324.458} C_VEL
LIN {X 0,Y 124.339,Z 1146.924,A -85,B 0,C 180,E1 24336.562,E2 24336.562} C_VEL
LIN {X 0,Y 105.01,Z 1157.659,A -85,B 0,C 180,E1 24354.782,E2 24354.782} C_VEL
LIN {X 0,Y 97.628,Z 1162.358,A -85,B 0,C 180,E1 24371.934,E2 24371.934} C_VEL
LIN {X 0,Y 96.633,Z 1163.988,A -85,B 0,C 180,E1 24390.004,E2 24390.004} C_VEL
LIN {X 0,Y 97.626,Z 1162.377,A -85,B 0,C 180,E1 24408.075,E2 24408.075} C_VEL
LIN {X 0,Y 106.909,Z 1156.585,A -85,B 0,C 180,E1 24427.883,E2 24427.883} C_VEL
LIN {X 0,Y 128.188,Z 1144.741,A -85,B 0,C 180,E1 24445.78,E2 24445.78} C_VEL
LIN {X 0,Y 136.997,Z 1139.632,A -85,B 0,C 180,E1 24450.322,E2 24450.322} C_VEL
LIN {X 0,Y 119.856,Z 1136.821,A -85,B 0,C 180,E1 24479.997,E2 24479.997} C_VEL
LIN {X 0,Y 143.139,Z 1132.325,A -85,B 0,C 180,E1 24509.481,E2 24509.481} C_VEL
LIN {X 0,Y 143.621,Z 1132.629,A -85,B 0,C 180,E1 24510.585,E2 24510.585} C_VEL
LIN {X 0,Y 119.296,Z 1145.564,A -85,B 0,C 180,E1 24523.92,E2 24523.92} C_VEL
LIN {X 0,Y 102.205,Z 1153.842,A -85,B 0,C 180,E1 24543.608,E2 24543.608} C_VEL
LIN {X 0,Y 96.95,Z 1156.627,A -85,B 0,C 180,E1 24561.011,E2 24561.011} C_VEL
LIN {X 0,Y 96.816,Z 1156.953,A -85,B 0,C 180,E1 24569.996,E2 24569.996} C_VEL
LIN {X 0,Y 98.746,Z 1155.553,A -85,B 0,C 180,E1 24587.855,E2 24587.855} C_VEL
LIN {X 0,Y 110.518,Z 1149.806,A -85,B 0,C 180,E1 24608.057,E2 24608.057} C_VEL
LIN {X 0,Y 134.324,Z 1137.741,A -85,B 0,C 180,E1 24625.13,E2 24625.13} C_VEL
LIN {X 0,Y 146.832,Z 1130.649,A -85,B 0,C 180,E1 24630.532,E2 24630.532} C_VEL
LIN {X 0,Y 156.087,Z 1124.125,A -85,B 0,C 180,E1 24635.602,E2 24635.602} C_VEL
LIN {X 0,Y 166.032,Z 1116.913,A -85,B 0,C 180,E1 24640.068,E2 24640.068} C_VEL
LIN {X 0,Y 196.888,Z 1094.006,A -85,B 0,C 180,E1 24646.136,E2 24646.136} C_VEL
LIN {X 0,Y 225.297,Z 1067.499,A -85,B 0,C 180,E1 24650.091,E2 24650.091} C_VEL
LIN {X 0,Y 232.789,Z 1059.43,A -85,B 0,C 180,E1 24650.996,E2 24650.996} C_VEL
LIN {X 0,Y 234.32,Z 1056.08,A -85,B 0,C 180,E1 24656.297,E2 24656.297} C_VEL
LIN {X 0,Y 234.402,Z 1056.152,A -85,B 0,C 180,E1 24660.002,E2 24660.002} C_VEL
LIN {X 0,Y 232.677,Z 1059.967,A -85,B 0,C 180,E1 24664.955,E2 24664.955} C_VEL
LIN {X 0,Y 202.65,Z 1090.101,A -85,B 0,C 180,E1 24668.923,E2 24668.923} C_VEL
LIN {X 0,Y 168.887,Z 1116.823,A -85,B 0,C 180,E1 24675.29,E2 24675.29} C_VEL
LIN {X 0,Y 137.493,Z 1136.775,A -85,B 0,C 180,E1 24684.705,E2 24684.705} C_VEL
LIN {X 0,Y 109.427,Z 1151.816,A -85,B 0,C 180,E1 24700.451,E2 24700.451} C_VEL
LIN {X 0,Y 93.324,Z 1160.099,A -85,B 0,C 180,E1 24720.879,E2 24720.879} C_VEL
LIN {X 0,Y 88.541,Z 1163.268,A -85,B 0,C 180,E1 24740.158,E2 24740.158} C_VEL
LIN {X 0,Y 88.709,Z 1163.7,A -85,B 0,C 180,E1 24750.005,E2 24750.005} C_VEL
LIN {X 0,Y 90.001,Z 1162.085,A -85,B 0,C 180,E1 24769.667,E2 24769.667} C_VEL
LIN {X 0,Y 102.998,Z 1155.116,A -85,B 0,C 180,E1 24793.574,E2 24793.574} C_VEL
LIN {X 0,Y 125.673,Z 1143.419,A -85,B 0,C 180,E1 24809.944,E2 24809.944} C_VEL
LIN {X 0,Y 126.933,Z 1142.346,A -85,B 0,C 180,E1 24811.501,E2 24811.501} C_VEL
LIN {X 0,Y 114.293,Z 1138.927,A -85,B 0,C 180,E1 24847.608,E2 24847.608} C_VEL
LIN {X 0,Y 134.142,Z 1135.656,A -85,B 0,C 180,E1 24869.476,E2 24869.476} C_VEL
LIN {X 0,Y 111.393,Z 1146.96,A -85,B 0,C 180,E1 24882.803,E2 24882.803} C_VEL
LIN {X 0,Y 95.093,Z 1154.133,A -85,B 0,C 180,E1 24901.461,E2 24901.461} C_VEL
LIN {X 0,Y 89.116,Z 1156.916,A -85,B 0,C 180,E1 24920.213,E2 24920.213} C_VEL
LIN {X 0,Y 88.918,Z 1157.241,A -85,B 0,C 180,E1 24929.995,E2 24929.995} C_VEL
LIN {X 0,Y 91.195,Z 1155.843,A -85,B 0,C 180,E1 24949.39,E2 24949.39} C_VEL
LIN {X 0,Y 104.289,Z 1150.099,A -85,B 0,C 180,E1 24970.789,E2 24970.789} C_VEL
LIN {X 0,Y 129.878,Z 1138.035,A -85,B 0,C 180,E1 24988.052,E2 24988.052} C_VEL
LIN {X 0,Y 162.114,Z 1119.538,A -85,B 0,C 180,E1 24999.059,E2 24999.059} C_VEL
LIN {X 0,Y 166.032,Z 1116.913,A -85,B 0,C 180,E1 25000.068,E2 25000.068} C_VEL
LIN {X 0,Y 176.607,Z 1108.968,A -85,B 0,C 180,E1 25003.935,E2 25003.935} C_VEL
LIN {X 0,Y 186.01,Z 1101.515,A -85,B 0,C 180,E1 25006.962,E2 25006.962} C_VEL
LIN {X 0,Y 187.597,Z 1100.304,A -85,B 0,C 180,E1 25007.244,E2 25007.244} C_VEL
LIN {X 0,Y 218.837,Z 1073.116,A -85,B 0,C 180,E1 25011.516,E2 25011.516} C_VEL
LIN {X 0,Y 227.24,Z 1064.524,A -85,B 0,C 180,E1 25012.433,E2 25012.433} C_VEL
LIN {X 0,Y 228.89,Z 1062.007,A -85,B 0,C 180,E1 25016.209,E2 25016.209} C_VEL
LIN {X 0,Y 228.999,Z 1062.059,A -85,B 0,C 180,E1 25020.002,E2 25020.002} C_VEL
LIN {X 0,Y 227.543,Z 1064.592,A -85,B 0,C 180,E1 25023.524,E2 25023.524} C_VEL
LIN {X 0,Y 198.334,Z 1092.498,A -85,B 0,C 180,E1 25027.061,E2 25027.061} C_VEL
LIN {X 0,Y 166.915,Z 1116.511,A -85,B 0,C 180,E1 25032.571,E2 25032.571} C_VEL
LIN {X 0,Y 134.239,Z 1136.478,A -85,B 0,C 180,E1 25041.505,E2 25041.505} C_VEL
LIN {X 0,Y 104.093,Z 1151.591,A -85,B 0,C 180,E1 25057.127,E2 25057.127} C_VEL
LIN {X 0,Y 86.325,Z 1159.803,A -85,B 0,C 180,E1 25078.257,E2 25078.257} C_VEL
LIN {X 0,Y 80.668,Z 1162.977,A -85,B 0,C 180,E1 25099.187,E2 25099.187} C_VEL
LIN {X 0,Y 80.775,Z 1163.411,A -85,B 0,C 180,E1 25110.005,E2 25110.005} C_VEL
LIN {X 0,Y 82.439,Z 1161.791,A -85,B 0,C 180,E1 25131.557,E2 25131.557} C_VEL
LIN {X 0,Y 95.25,Z 1155.645,A -85,B 0,C 180,E1 25154.883,E2 25154.883} C_VEL
LIN {X 0,Y 116.247,Z 1145.877,A -85,B 0,C 180,E1 25170.586,E2 25170.586} C_VEL
LIN {X 0,Y 117.761,Z 1144.79,A -85,B 0,C 180,E1 25172.134,E2 25172.134} C_VEL
LIN {X 0,Y 107.428,Z 1141.483,A -85,B 0,C 180,E1 25209.365,E2 25209.365} C_VEL
LIN {X 0,Y 124.593,Z 1138.903,A -85,B 0,C 180,E1 25229.077,E2 25229.077} C_VEL
LIN {X 0,Y 98.311,Z 1150.453,A -85,B 0,C 180,E1 25246.121,E2 25246.121} C_VEL
LIN {X 0,Y 83.689,Z 1156.17,A -85,B 0,C 180,E1 25268.781,E2 25268.781} C_VEL
LIN {X 0,Y 81.004,Z 1157.528,A -85,B 0,C 180,E1 25289.995,E2 25289.995} C_VEL
LIN {X 0,Y 83.7,Z 1156.134,A -85,B 0,C 180,E1 25311.206,E2 25311.206} C_VEL
LIN {X 0,Y 98.336,Z 1150.39,A -85,B 0,C 180,E1 25333.853,E2 25333.853} C_VEL
LIN {X 0,Y 126.052,Z 1138.21,A -85,B 0,C 180,E1 25351.291,E2 25351.291} C_VEL
LIN {X 0,Y 159.411,Z 1119.845,A -85,B 0,C 180,E1 25361.765,E2 25361.765} C_VEL
LIN {X 0,Y 187.597,Z 1100.304,A -85,B 0,C 180,E1 25367.244,E2 25367.244} C_VEL
LIN {X 0,Y 198.705,Z 1090.972,A -85,B 0,C 180,E1 25370.168,E2 25370.168} C_VEL
LIN {X 0,Y 209.835,Z 1080.981,A -85,B 0,C 180,E1 25372.73,E2 25372.73} C_VEL
LIN {X 0,Y 222.668,Z 1068.623,A -85,B 0,C 180,E1 25374.257,E2 25374.257} C_VEL
LIN {X 0,Y 223.261,Z 1067.726,A -85,B 0,C 180,E1 25376.114,E2 25376.114} C_VEL
LIN {X 0,Y 222.893,Z 1068.508,A -85,B 0,C 180,E1 25381.193,E2 25381.193} C_VEL
LIN {X 0,Y 221.971,Z 1069.66,A -85,B 0,C 180,E1 25381.971,E2 25381.971} C_VEL
LIN {X 0,Y 190.196,Z 1098.121,A -85,B 0,C 180,E1 25385.686,E2 25385.686} C_VEL
LIN {X 0,Y 154.735,Z 1122.953,A -85,B 0,C 180,E1 25391.905,E2 25391.905} C_VEL
LIN {X 0,Y 120.636,Z 1141.649,A -85,B 0,C 180,E1 25402.12,E2 25402.12} C_VEL
LIN {X 0,Y 90.532,Z 1154.967,A -85,B 0,C 180,E1 25420.561,E2 25420.561} C_VEL
LIN {X 0,Y 75.011,Z 1161.477,A -85,B 0,C 180,E1 25446.196,E2 25446.196} C_VEL
LIN {X 0,Y 72.838,Z 1163.123,A -85,B 0,C 180,E1 25470.006,E2 25470.006} C_VEL
LIN {X 0,Y 75.01,Z 1161.498,A -85,B 0,C 180,E1 25493.817,E2 25493.817} C_VEL
LIN {X 0,Y 90.472,Z 1155.015,A -85,B 0,C 180,E1 25519.439,E2 25519.439} C_VEL
LIN {X 0,Y 104.741,Z 1148.972,A -85,B 0,C 180,E1 25530.161,E2 25530.161} C_VEL
LIN {X 0,Y 108.219,Z 1147.099,A -85,B 0,C 180,E1 25533.214,E2 25533.214} C_VEL
LIN {X 0,Y 103.89,Z 1143.352,A -85,B 0,C 180,E1 25576.941,E2 25576.941} C_VEL
LIN {X 0,Y 113.923,Z 1142.004,A -85,B 0,C 180,E1 25587.714,E2 25587.714} C_VEL
LIN {X 0,Y 111.045,Z 1143.539,A -85,B 0,C 180,E1 25590.321,E2 25590.321} C_VEL
LIN {X 0,Y 84.633,Z 1153.568,A -85,B 0,C 180,E1 25611.226,E2 25611.226} C_VEL
LIN {X 0,Y 73.499,Z 1157.494,A -85,B 0,C 180,E1 25638.106,E2 25638.106} C_VEL
LIN {X 0,Y 73.107,Z 1157.816,A -85,B 0,C 180,E1 25649.994,E2 25649.994} C_VEL
LIN {X 0,Y 76.332,Z 1156.424,A -85,B 0,C 180,E1 25673.368,E2 25673.368} C_VEL
LIN {X 0,Y 92.685,Z 1150.683,A -85,B 0,C 180,E1 25697.312,E2 25697.312} C_VEL
LIN {X 0,Y 122.373,Z 1138.505,A -85,B 0,C 180,E1 25714.614,E2 25714.614} C_VEL
LIN {X 0,Y 157.058,Z 1120.154,A -85,B 0,C 180,E1 25724.583,E2 25724.583} C_VEL
LIN {X 0,Y 190.631,Z 1097.098,A -85,B 0,C 180,E1 25730.339,E2 25730.339} C_VEL
LIN {X 0,Y 209.835,Z 1080.981,A -85,B 0,C 180,E1 25732.73,E2 25732.73} C_VEL
LIN {X 0,Y 214.672,Z 1076.375,A -85,B 0,C 180,E1 25734.269,E2 25734.269} C_VEL
LIN {X 0,Y 217.292,Z 1073.508,A -85,B 0,C 180,E1 25737.45,E2 25737.45} C_VEL
LIN {X 0,Y 217.434,Z 1073.386,A -85,B 0,C 180,E1 25738.299,E2 25738.299} C_VEL
LIN {X 0,Y 217.613,Z 1073.407,A -85,B 0,C 180,E1 25740.002,E2 25740.002} C_VEL
LIN {X 0,Y 208.229,Z 1082.213,A -85,B 0,C 180,E1 25741.155,E2 25741.155} C_VEL
LIN {X 0,Y 174.7,Z 1108.748,A -85,B 0,C 180,E1 25745.238,E2 25745.238} C_VEL
LIN {X 0,Y 139.287,Z 1130.534,A -85,B 0,C 180,E1 25751.957,E2 25751.957} C_VEL
LIN {X 0,Y 106.808,Z 1146.219,A -85,B 0,C 180,E1 25762.87,E2 25762.87} C_VEL
LIN {X 0,Y 80.474,Z 1156.464,A -85,B 0,C 180,E1 25781.191,E2 25781.191} C_VEL
LIN {X 0,Y 67.71,Z 1161.183,A -85,B 0,C 180,E1 25803.44,E2 25803.44} C_VEL
LIN {X 0,Y 64.898,Z 1162.834,A -85,B 0,C 180,E1 25830.006,E2 25830.006} C_VEL
LIN {X 0,Y 67.684,Z 1161.204,A -85,B 0,C 180,E1 25856.584,E2 25856.584} C_VEL
LIN {X 0,Y 84.985,Z 1154.847,A -85,B 0,C 180,E1 25883.304,E2 25883.304} C_VEL
LIN {X 0,Y 99.106,Z 1149.215,A -85,B 0,C 180,E1 25893.944,E2 25893.944} C_VEL
LIN {X 0,Y 96.699,Z 1145.683,A -85,B 0,C 180,E1 25938.243,E2 25938.243} C_VEL
LIN {X 0,Y 104.246,Z 1144.748,A -85,B 0,C 180,E1 25946.985,E2 25946.985} C_VEL
LIN {X 0,Y 103.319,Z 1145.296,A -85,B 0,C 180,E1 25948.434,E2 25948.434} C_VEL
LIN {X 0,Y 78.522,Z 1153.858,A -85,B 0,C 180,E1 25967.546,E2 25967.546} C_VEL
LIN {X 0,Y 65.739,Z 1157.783,A -85,B 0,C 180,E1 25996.678,E2 25996.678} C_VEL
LIN {X 0,Y 65.19,Z 1158.104,A -85,B 0,C 180,E1 26009.994,E2 26009.994} C_VEL
LIN {X 0,Y 72.267,Z 1155.734,A -85,B 0,C 180,E1 26043.083,E2 26043.083} C_VEL
LIN {X 0,Y 92.401,Z 1149.234,A -85,B 0,C 180,E1 26065.01,E2 26065.01} C_VEL
LIN {X 0,Y 121.624,Z 1137.664,A -85,B 0,C 180,E1 26079,E2 26079} C_VEL
LIN {X 0,Y 155.103,Z 1120.462,A -85,B 0,C 180,E1 26087.466,E2 26087.466} C_VEL
LIN {X 0,Y 190.038,Z 1096.956,A -85,B 0,C 180,E1 26092.802,E2 26092.802} C_VEL
LIN {X 0,Y 216.521,Z 1074.296,A -85,B 0,C 180,E1 26095.642,E2 26095.642} C_VEL
LIN {X 0,Y 217.496,Z 1073.357,A -85,B 0,C 180,E1 26096.01,E2 26096.01} C_VEL
LIN {X 0,Y 217.434,Z 1073.386,A -85,B 0,C 180,E1 26098.299,E2 26098.299} C_VEL
LIN {X 0,Y 215.183,Z 1075.586,A -85,B 0,C 180,E1 26099.247,E2 26099.247} C_VEL
LIN {X 0,Y 205.553,Z 1084.199,A -85,B 0,C 180,E1 26099.467,E2 26099.467} C_VEL
LIN {X 0,Y 200.115,Z 1088.817,A -85,B 0,C 180,E1 26099.633,E2 26099.633} C_VEL
LIN {X 0,Y 165.009,Z 1114.479,A -85,B 0,C 180,E1 26103.764,E2 26103.764} C_VEL
LIN {X 0,Y 128.369,Z 1135.025,A -85,B 0,C 180,E1 26110.768,E2 26110.768} C_VEL
LIN {X 0,Y 93.547,Z 1149.892,A -85,B 0,C 180,E1 26123.423,E2 26123.423} C_VEL
LIN {X 0,Y 66.774,Z 1158.911,A -85,B 0,C 180,E1 26147.144,E2 26147.144} C_VEL
LIN {X 0,Y 57.264,Z 1162.103,A -85,B 0,C 180,E1 26174.675,E2 26174.675} C_VEL
LIN {X 0,Y 56.953,Z 1162.545,A -85,B 0,C 180,E1 26190.007,E2 26190.007} C_VEL
LIN {X 0,Y 60.55,Z 1160.91,A -85,B 0,C 180,E1 26220.016,E2 26220.016} C_VEL
LIN {X 0,Y 80.343,Z 1154.55,A -85,B 0,C 180,E1 26248.011,E2 26248.011} C_VEL
LIN {X 0,Y 87.955,Z 1151.918,A -85,B 0,C 180,E1 26253.336,E2 26253.336} C_VEL
LIN {X 0,Y 89.633,Z 1151.111,A -85,B 0,C 180,E1 26255.353,E2 26255.353} C_VEL
LIN {X 0,Y 94.194,Z 1147.397,A -85,B 0,C 180,E1 26305.651,E2 26305.651} C_VEL
LIN {X 0,Y 91.365,Z 1148.493,A -85,B 0,C 180,E1 26308.582,E2 26308.582} C_VEL
LIN {X 0,Y 68.627,Z 1155.297,A -85,B 0,C 180,E1 26328.547,E2 26328.547} C_VEL
LIN {X 0,Y 58.036,Z 1158.072,A -85,B 0,C 180,E1 26354.87,E2 26354.87} C_VEL
LIN {X 0,Y 57.301,Z 1158.39,A -85,B 0,C 180,E1 26369.993,E2 26369.993} C_VEL
LIN {X 0,Y 61.983,Z 1157.007,A -85,B 0,C 180,E1 26399.239,E2 26399.239} C_VEL
LIN {X 0,Y 81.868,Z 1151.478,A -85,B 0,C 180,E1 26425.031,E2 26425.031} C_VEL
LIN {X 0,Y 115.676,Z 1139.365,A -85,B 0,C 180,E1 26441.608,E2 26441.608} C_VEL
LIN {X 0,Y 153.554,Z 1120.77,A -85,B 0,C 180,E1 26450.405,E2 26450.405} C_VEL
LIN {X 0,Y 189.922,Z 1096.715,A -85,B 0,C 180,E1 26455.302,E2 26455.302} C_VEL
LIN {X 0,Y 211.63,Z 1078.739,A -85,B 0,C 180,E1 26457.439,E2 26457.439} C_VEL
LIN {X 0,Y 211.667,Z 1078.739,A -85,B 0,C 180,E1 26458.435,E2 26458.435} C_VEL
LIN {X 0,Y 200.115,Z 1088.817,A -85,B 0,C 180,E1 26459.633,E2 26459.633} C_VEL
LIN {X 0,Y 193.519,Z 1094.097,A -85,B 0,C 180,E1 26459.228,E2 26459.228} C_VEL
LIN {X 0,Y 182.472,Z 1102.071,A -85,B 0,C 180,E1 26457.041,E2 26457.041} C_VEL
LIN {X 0,Y 148.78,Z 1123.034,A -85,B 0,C 180,E1 26452.845,E2 26452.845} C_VEL
LIN {X 0,Y 113.383,Z 1139.66,A -85,B 0,C 180,E1 26445.492,E2 26445.492} C_VEL
LIN {X 0,Y 81.516,Z 1150.655,A -85,B 0,C 180,E1 26432.496,E2 26432.496} C_VEL
LIN {X 0,Y 55.137,Z 1157.298,A -85,B 0,C 180,E1 26403.305,E2 26403.305} C_VEL
LIN {X 0,Y 49.379,Z 1158.678,A -85,B 0,C 180,E1 26369.992,E2 26369.992} C_VEL
LIN {X 0,Y 56.79,Z 1156.922,A -85,B 0,C 180,E1 26333.095,E2 26333.095} C_VEL
LIN {X 0,Y 84.161,Z 1149.89,A -85,B 0,C 180,E1 26305.89,E2 26305.89} C_VEL
LIN {X 0,Y 82.361,Z 1149.901,A -85,B 0,C 180,E1 26301.565,E2 26301.565} C_VEL
LIN {X 0,Y 80.499,Z 1152.851,A -85,B 0,C 180,E1 26256.612,E2 26256.612} C_VEL
LIN {X 0,Y 61.045,Z 1158.646,A -85,B 0,C 180,E1 26238.092,E2 26238.092} C_VEL
LIN {X 0,Y 49.546,Z 1161.823,A -85,B 0,C 180,E1 26207.803,E2 26207.803} C_VEL
LIN {X 0,Y 49.006,Z 1162.256,A -85,B 0,C 180,E1 26190.008,E2 26190.008} C_VEL
LIN {X 0,Y 53.702,Z 1160.593,A -85,B 0,C 180,E1 26155.683,E2 26155.683} C_VEL
LIN {X 0,Y 76.31,Z 1154.214,A -85,B 0,C 180,E1 26126.774,E2 26126.774} C_VEL
LIN {X 0,Y 111.785,Z 1141.468,A -85,B 0,C 180,E1 26110.901,E2 26110.901} C_VEL
LIN {X 0,Y 151.575,Z 1122.016,A -85,B 0,C 180,E1 26102.704,E2 26102.704} C_VEL
LIN {X 0,Y 188.413,Z 1097.852,A -85,B 0,C 180,E1 26098.305,E2 26098.305} C_VEL
LIN {X 0,Y 191.841,Z 1095.19,A -85,B 0,C 180,E1 26097.947,E2 26097.947} C_VEL
LIN {X 0,Y 182.472,Z 1102.071,A -85,B 0,C 180,E1 26097.041,E2 26097.041} C_VEL
LIN {X 0,Y 167.832,Z 1111.845,A -85,B 0,C 180,E1 26096.846,E2 26096.846} C_VEL
LIN {X 0,Y 152.81,Z 1120.748,A -85,B 0,C 180,E1 26096.56,E2 26096.56} C_VEL
LIN {X 0,Y 115.19,Z 1138.558,A -85,B 0,C 180,E1 26090.33,E2 26090.33} C_VEL
LIN {X 0,Y 80.977,Z 1150.12,A -85,B 0,C 180,E1 26079.201,E2 26079.201} C_VEL
LIN {X 0,Y 57.579,Z 1155.838,A -85,B 0,C 180,E1 26062.072,E2 26062.072} C_VEL
LIN {X 0,Y 42.892,Z 1158.631,A -85,B 0,C 180,E1 26030.662,E2 26030.662} C_VEL
LIN {X 0,Y 41.457,Z 1158.967,A -85,B 0,C 180,E1 26009.99,E2 26009.99} C_VEL
LIN {X 0,Y 48.656,Z 1157.62,A -85,B 0,C 180,E1 25971.499,E2 25971.499} C_VEL
LIN {X 0,Y 75.234,Z 1151.767,A -85,B 0,C 180,E1 25943.726,E2 25943.726} C_VEL
LIN {X 0,Y 70.934,Z 1154.286,A -85,B 0,C 180,E1 25899.328,E2 25899.328} C_VEL
LIN {X 0,Y 66.874,Z 1155.607,A -85,B 0,C 180,E1 25894.928,E2 25894.928} C_VEL
LIN {X 0,Y 47.208,Z 1160.32,A -85,B 0,C 180,E1 25869.913,E2 25869.913} C_VEL
LIN {X 0,Y 41.056,Z 1161.967,A -85,B 0,C 180,E1 25830.01,E2 25830.01} C_VEL
LIN {X 0,Y 47.222,Z 1160.297,A -85,B 0,C 180,E1 25790.124,E2 25790.124} C_VEL
LIN {X 0,Y 72.969,Z 1153.913,A -85,B 0,C 180,E1 25760.986,E2 25760.986} C_VEL
LIN {X 0,Y 110.516,Z 1141.165,A -85,B 0,C 180,E1 25746.672,E2 25746.672} C_VEL
LIN {X 0,Y 151.41,Z 1121.703,A -85,B 0,C 180,E1 25739.591,E2 25739.591} C_VEL
LIN {X 0,Y 161.172,Z 1116.008,A -85,B 0,C 180,E1 25738.405,E2 25738.405} C_VEL
LIN {X 0,Y 162.755,Z 1115.059,A -85,B 0,C 180,E1 25737.677,E2 25737.677} C_VEL
LIN {X 0,Y 152.81,Z 1120.748,A -85,B 0,C 180,E1 25736.56,E2 25736.56} C_VEL
LIN {X 0,Y 137.29,Z 1128.87,A -85,B 0,C 180,E1 25736.129,E2 25736.129} C_VEL
LIN {X 0,Y 121.3,Z 1135.935,A -85,B 0,C 180,E1 25735.538,E2 25735.538} C_VEL
LIN {X 0,Y 85.383,Z 1148.553,A -85,B 0,C 180,E1 25727.228,E2 25727.228} C_VEL
LIN {X 0,Y 53.025,Z 1156.131,A -85,B 0,C 180,E1 25708.928,E2 25708.928} C_VEL
LIN {X 0,Y 35.553,Z 1158.921,A -85,B 0,C 180,E1 25675.194,E2 25675.194} C_VEL
LIN {X 0,Y 33.533,Z 1159.255,A -85,B 0,C 180,E1 25649.988,E2 25649.988} C_VEL
LIN {X 0,Y 42.698,Z 1157.911,A -85,B 0,C 180,E1 25604.815,E2 25604.815} C_VEL
LIN {X 0,Y 65.205,Z 1153.702,A -85,B 0,C 180,E1 25581.728,E2 25581.728} C_VEL
LIN {X 0,Y 61.731,Z 1155.61,A -85,B 0,C 180,E1 25542.456,E2 25542.456} C_VEL
LIN {X 0,Y 60.23,Z 1156.195,A -85,B 0,C 180,E1 25539.246,E2 25539.246} C_VEL
LIN {X 0,Y 35.991,Z 1160.916,A -85,B 0,C 180,E1 25502.702,E2 25502.702} C_VEL
LIN {X 0,Y 33.1,Z 1161.678,A -85,B 0,C 180,E1 25470.012,E2 25470.012} C_VEL
LIN {X 0,Y 41.323,Z 1160.001,A -85,B 0,C 180,E1 25422.89,E2 25422.89} C_VEL
LIN {X 0,Y 70.436,Z 1153.614,A -85,B 0,C 180,E1 25394.704,E2 25394.704} C_VEL
LIN {X 0,Y 109.862,Z 1140.863,A -85,B 0,C 180,E1 25382.37,E2 25382.37} C_VEL
LIN {X 0,Y 136.333,Z 1129.311,A -85,B 0,C 180,E1 25378.189,E2 25378.189} C_VEL
LIN {X 0,Y 136.374,Z 1129.269,A -85,B 0,C 180,E1 25377.71,E2 25377.71} C_VEL
LIN {X 0,Y 121.3,Z 1135.935,A -85,B 0,C 180,E1 25375.538,E2 25375.538} C_VEL
LIN {X 0,Y 104.959,Z 1142.201,A -85,B 0,C 180,E1 25374.756,E2 25374.756} C_VEL
LIN {X 0,Y 88.371,Z 1147.567,A -85,B 0,C 180,E1 25373.714,E2 25373.714} C_VEL
LIN {X 0,Y 49.357,Z 1156.424,A -85,B 0,C 180,E1 25356.951,E2 25356.951} C_VEL
LIN {X 0,Y 28.551,Z 1159.211,A -85,B 0,C 180,E1 25322.011,E2 25322.011} C_VEL
LIN {X 0,Y 25.626,Z 1159.542,A -85,B 0,C 180,E1 25289.984,E2 25289.984} C_VEL
LIN {X 0,Y 37.483,Z 1158.202,A -85,B 0,C 180,E1 25236.089,E2 25236.089} C_VEL
LIN {X 0,Y 52.33,Z 1155.934,A -85,B 0,C 180,E1 25220.833,E2 25220.833} C_VEL
LIN {X 0,Y 55.125,Z 1155.427,A -85,B 0,C 180,E1 25217.822,E2 25217.822} C_VEL
LIN {X 0,Y 52.902,Z 1156.722,A -85,B 0,C 180,E1 25185.491,E2 25185.491} C_VEL
LIN {X 0,Y 48.232,Z 1157.755,A -85,B 0,C 180,E1 25180.376,E2 25180.376} C_VEL
LIN {X 0,Y 27.599,Z 1160.947,A -85,B 0,C 180,E1 25143.289,E2 25143.289} C_VEL
LIN {X 0,Y 25.149,Z 1161.389,A -85,B 0,C 180,E1 25110.016,E2 25110.016} C_VEL
LIN {X 0,Y 36.281,Z 1159.705,A -85,B 0,C 180,E1 25053.438,E2 25053.438} C_VEL
LIN {X 0,Y 68.807,Z 1153.315,A -85,B 0,C 180,E1 25028.048,E2 25028.048} C_VEL
LIN {X 0,Y 110.077,Z 1140.472,A -85,B 0,C 180,E1 25018.016,E2 25018.016} C_VEL
LIN {X 0,Y 88.371,Z 1147.567,A -85,B 0,C 180,E1 25013.714,E2 25013.714} C_VEL
LIN {X 0,Y 71.514,Z 1152.039,A -85,B 0,C 180,E1 25012.219,E2 25012.219} C_VEL
LIN {X 0,Y 54.475,Z 1155.452,A -85,B 0,C 180,E1 25009.875,E2 25009.875} C_VEL
LIN {X 0,Y 22.2,Z 1159.501,A -85,B 0,C 180,E1 24972.979,E2 24972.979} C_VEL
LIN {X 0,Y 17.698,Z 1159.831,A -85,B 0,C 180,E1 24929.977,E2 24929.977} C_VEL
LIN {X 0,Y 39.935,Z 1157.682,A -85,B 0,C 180,E1 24858.55,E2 24858.55} C_VEL
LIN {X 0,Y 45.417,Z 1156.983,A -85,B 0,C 180,E1 24852.513,E2 24852.513} C_VEL
LIN {X 0,Y 44.293,Z 1157.728,A -85,B 0,C 180,E1 24830.15,E2 24830.15} C_VEL
LIN {X 0,Y 32.529,Z 1159.436,A -85,B 0,C 180,E1 24818.618,E2 24818.618} C_VEL
LIN {X 0,Y 17.18,Z 1161.099,A -85,B 0,C 180,E1 24750.023,E2 24750.023} C_VEL
LIN {X 0,Y 32.523,Z 1159.41,A -85,B 0,C 180,E1 24681.425,E2 24681.425} C_VEL
LIN {X 0,Y 72.58,Z 1151.961,A -85,B 0,C 180,E1 24660.006,E2 24660.006} C_VEL
LIN {X 0,Y 81.632,Z 1149.569,A -85,B 0,C 180,E1 24658.069,E2 24658.069} C_VEL
LIN {X 0,Y 54.475,Z 1155.452,A -85,B 0,C 180,E1 24649.875,E2 24649.875} C_VEL
LIN {X 0,Y 41.761,Z 1157.449,A -85,B 0,C 180,E1 24646.664,E2 24646.664} C_VEL
LIN {X 0,Y 22.247,Z 1159.423,A -85,B 0,C 180,E1 24640.187,E2 24640.187} C_VEL
LIN {X 0,Y 20.29,Z 1159.543,A -85,B 0,C 180,E1 24637.472,E2 24637.472} C_VEL
LIN {X 0,Y 9.789,Z 1160.118,A -85,B 0,C 180,E1 24569.959,E2 24569.959} C_VEL
LIN {X 0,Y 35.09,Z 1158.312,A -85,B 0,C 180,E1 24488.66,E2 24488.66} C_VEL
LIN {X 0,Y 36.283,Z 1158.228,A -85,B 0,C 180,E1 24484.794,E2 24484.794} C_VEL
LIN {X 0,Y 35.998,Z 1158.414,A -85,B 0,C 180,E1 24477.616,E2 24477.616} C_VEL
LIN {X 0,Y 16.668,Z 1160.361,A -85,B 0,C 180,E1 24455.345,E2 24455.345} C_VEL
LIN {X 0,Y 9.209,Z 1160.809,A -85,B 0,C 180,E1 24390.044,E2 24390.044} C_VEL
LIN {X 0,Y 30.505,Z 1159.113,A -85,B 0,C 180,E1 24307.025,E2 24307.025} C_VEL
LIN {X 0,Y 50.845,Z 1156.203,A -85,B 0,C 180,E1 24298.089,E2 24298.089} C_VEL
LIN {X 0,Y 20.29,Z 1159.543,A -85,B 0,C 180,E1 24277.472,E2 24277.472} C_VEL
LIN {X 0,Y 9.165,Z 1160.187,A -85,B 0,C 180,E1 24263.465,E2 24263.465} C_VEL
LIN {X 0,Y 4.057,Z 1160.355,A -85,B 0,C 180,E1 24133.712,E2 24133.712} C_VEL
LIN {X 0,Y 8.195,Z 1160.299,A -85,B 0,C 180,E1 24119.95,E2 24119.95} C_VEL
LIN {X 0,Y 1.227,Z 1160.519,A -85,B 0,C 180,E1 24030.329,E2 24030.329} C_VEL
LIN {X 0,Y 8.444,Z 1160.288,A -85,B 0,C 180,E1 23940.048,E2 23940.048} C_VEL
LIN {X 0,Y 1.858,Z 1160.406,A -85,B 0,C 180,E1 23849.783,E2 23849.783} C_VEL
LIN {X 0,Y 4.057,Z 1160.355,A -85,B 0,C 180,E1 23773.712,E2 23773.712} C_VEL
LIN {X 0,Y 5.939,Z 1162.355,A -85,B 0,C 180,E1 23764.945,E2 23764.945} C_VEL
LIN {X 0,Y 5.939,Z 1180,A -85,B 0,C 180,E1 23764.945,E2 23764.945} C_VEL
LIN {X 0,Y 5.939,Z 1180,A -85,B 0,C 180,E1 23764.945,E2 23764.945}

